// TIA Portal V17 program export: 1 tag tables, 0 data types, 1 data blocks, 4 code blocks (in call order from the OBs), 0 instance data blocks

VAR_GLOBAL   // PLC tag table "Default tag table"
   vystup2 AT %Q1.0 : Bool;
   vystup1 AT %Q0.0 : Bool;
   Tag_1 AT %MW50 : Int;
   Tag_2 AT %MW52 : Word;
   Tag_3 AT %MW54 : Int;
   Tag_4 AT %MW56 : Word;
   vstup2 AT %I20.0 : Bool;
   vstup1 AT %I20.1 : Bool;
   xxx AT %I20.2 : Bool;
END_VAR

DATA_BLOCK "Data_block_1"   // DB1
VERSION : 0.1
// stored: AutoNumber true, IsOnlyStoredInLoadMemory false, IsWriteProtectedInAS false
BEGIN
END_DATA_BLOCK

ORGANIZATION_BLOCK "Main"   // OB1, LAD, ProgramCycle
TITLE = "Main Program Sweep (Cycle)"
VERSION : 0.1
// stored: IsIECCheckEnabled false
   VAR_TEMP
      OB1_EV_CLASS : Byte;   // Bits 0-3 = 1 (Coming event), Bits 4-7 = 1 (Event class 1)
      OB1_SCAN_1 : Byte;   // 1 (Cold restart scan 1 of OB 1), 3 (Scan 2-n of OB 1)
      OB1_PRIORITY : Byte;   // Priority of OB Execution
      OB1_OB_NUMBR : Byte;   // 1 (Organization block 1, OB1)
      OB1_RESERVED_1 : Byte;   // Reserved for system
      OB1_RESERVED_2 : Byte;   // Reserved for system
      OB1_PREV_CYCLE : Int;   // Cycle time of previous OB1 scan (milliseconds)
      OB1_MIN_CYCLE : Int;   // Minimum cycle time of OB1 (milliseconds)
      OB1_MAX_CYCLE : Int;   // Maximum cycle time of OB1 (milliseconds)
      OB1_DATE_TIME : Date_And_Time;   // Date and time OB1 started
   END_VAR
BEGIN

REGION Network 1
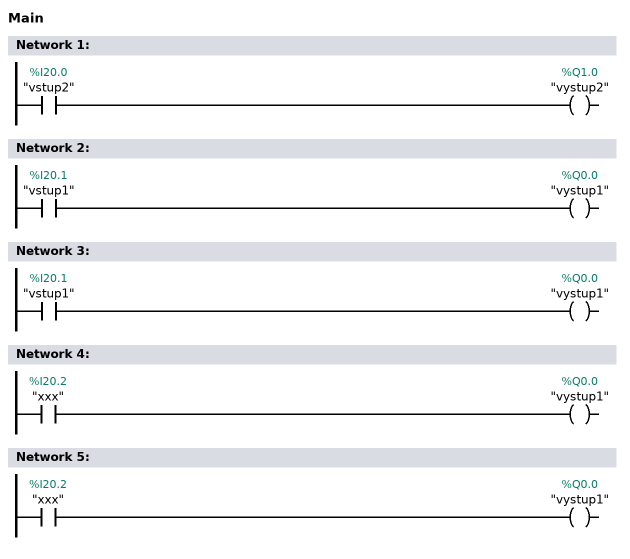
   RUNG wire#powerrail
      Contact( "vstup2" )
      Coil( "vystup2" )
   END_RUNG
   // the same network as SCL:
   "vystup2" := "vstup2";
END_REGION

REGION Network 2
   RUNG wire#powerrail
      Contact( "vstup1" )
      Coil( "vystup1" )
   END_RUNG
   // the same network as SCL:
   "vystup1" := "vstup1";
END_REGION

REGION Network 3
   RUNG wire#powerrail
      Contact( "vstup1" )
      Coil( "vystup1" )
   END_RUNG
   // the same network as SCL:
   "vystup1" := "vstup1";
END_REGION

REGION Network 4
   RUNG wire#powerrail
      Contact( "xxx" )
      Coil( "vystup1" )
   END_RUNG
   // the same network as SCL:
   "vystup1" := "xxx";
END_REGION

REGION Network 5
   RUNG wire#powerrail
      Contact( "xxx" )
      Coil( "vystup1" )
   END_RUNG
   // the same network as SCL:
   "vystup1" := "xxx";
END_REGION
END_ORGANIZATION_BLOCK

ORGANIZATION_BLOCK "RACK_FLT"   // OB86, LAD, RackOrStationFailure
TITLE = "Loss Of Rack Fault"
VERSION : 0.1
// stored: IsIECCheckEnabled false
   VAR_TEMP
      OB86_EV_CLASS : Byte;   // 16#38/39 Event class 3
      OB86_FLT_ID : Byte;   // 16#C1/C4/C5, Fault identification code
      OB86_PRIORITY : Byte;   // Priority of OB Execution
      OB86_OB_NUMBR : Byte;   // 86 (Organization block 86, OB86)
      OB86_RESERVED_1 : Byte;   // Reserved for system
      OB86_RESERVED_2 : Byte;   // Reserved for system
      OB86_MDL_ADDR : Word;   // Base address of IM module in rack with fault
      OB86_RACKS_FLTD : Array[0..31] of Bool;   // Racks in fault
      OB86_DATE_TIME : Date_And_Time;   // Date and time OB86 started
   END_VAR
BEGIN
END_ORGANIZATION_BLOCK

ORGANIZATION_BLOCK "SYNC_1"   // OB61, LAD, SynchronousCycle
TITLE = "DP Synchronous Interrupt"
VERSION : 0.1
// stored: IsIECCheckEnabled false
   VAR_TEMP
      OB61_EV_CLASS : Byte;   // Bits 0-3 = 1 (Coming event), Bits 4-7 = 1 (Event class 1)
      OB61_STRT_INF : Byte;   // OB 61 has started
      OB61_PRIORITY : Byte;   // Priority of OB Execution
      OB61_OB_NUMBR : Byte;   // 61 (Organization block 61, OB61)
      OB61_RESERVED_1 : Byte;   // Reserved for system
      OB61_RESERVED_2 : Byte;   // Reserved for system
      OB61_GC_VIOL : Bool;   // Lost Global Control of DP system
      OB61_FIRST : Bool;   // First Execution after startup or HALT
      OB61_MISSED_EXEC : Byte;   // Count of missed executions of OB61 since it was last scheduled
      OB61_DP_ID : Byte;   // DP master system ID of the synchronous DP system
      OB61_RESERVED_3 : Byte;   // Reserved for system
      OB61_RESERVED_4 : Word;   // Reserved for system
      OB61_DATE_TIME : Date_And_Time;   // Date and time OB61 started
   END_VAR
BEGIN

REGION Network 1
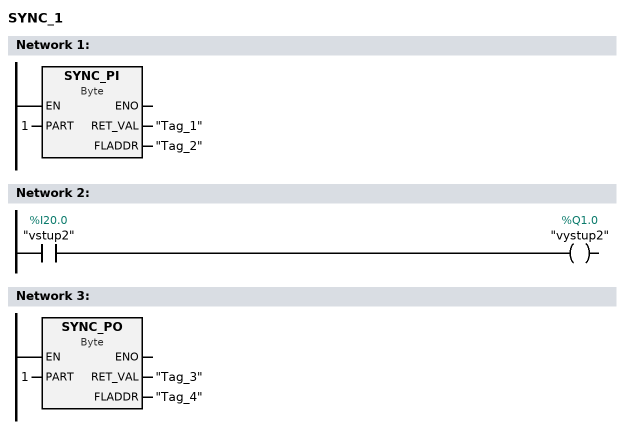
   RUNG wire#powerrail
      { S7_Templates := "value_type := Byte" } SYNC_PI(PART := 1, RET_VAL => "Tag_1", FLADDR => "Tag_2")
   END_RUNG
   // the same network as SCL:
   "Tag_1" := SYNC_PI(PART := 1, FLADDR => "Tag_2");
END_REGION

REGION Network 2
   RUNG wire#powerrail
      Contact( "vstup2" )
      Coil( "vystup2" )
   END_RUNG
   // the same network as SCL:
   "vystup2" := "vstup2";
END_REGION

REGION Network 3
   RUNG wire#powerrail
      { S7_Templates := "value_type := Byte" } SYNC_PO(PART := 1, RET_VAL => "Tag_3", FLADDR => "Tag_4")
   END_RUNG
   // the same network as SCL:
   "Tag_3" := SYNC_PO(PART := 1, FLADDR => "Tag_4");
END_REGION
END_ORGANIZATION_BLOCK

FUNCTION "Block_1" : Void
{ S7_Optimized_Access := 'FALSE' }
VERSION : 0.1

BEGIN
	"xxx" := "xxx";
END_FUNCTION
